Staubli VAL3: FC_InitMotion.pgx

program FC_InitMotion()
begin
  //this function is goiong to begin the synchronous motion
  $movejSyncBegin(mNomSpeed)
end
